// TIA Portal V19 export
FUNCTION "ValveMachine_PB_Connector" : Void   // FC157, LAD
TITLE = Collect push buttons for Valve Machine
// stored: Access Published, SetENOAutomatically false
   VAR_INPUT
      Enable : Bool;
      HMI_PB : "ValveMachine_PB";   // Push button from HMI a (e.g. MB1)
      LB_PB_Rest : Bool;
      LB_PB_Work : Bool;
      LB_PB_StartStop : Bool;
      Other_PB : "ValveMachine_PB";
   END_VAR
   VAR_OUTPUT
      PB : "ValveMachine_PB";
   END_VAR
BEGIN

REGION Network 1: Logical OR
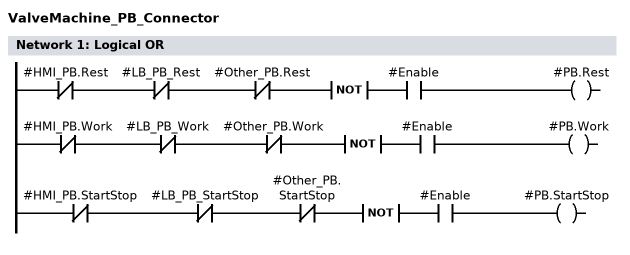
   RUNG wire#powerrail
      I_Contact( #HMI_PB.Rest )
      I_Contact( #LB_PB_Rest )
      I_Contact( #Other_PB.Rest )
      Not()
      Contact( #Enable )
      Coil( #PB.Rest )
   END_RUNG
   RUNG wire#powerrail
      I_Contact( #HMI_PB.Work )
      I_Contact( #LB_PB_Work )
      I_Contact( #Other_PB.Work )
      Not()
      Contact( #Enable )
      Coil( #PB.Work )
   END_RUNG
   RUNG wire#powerrail
      I_Contact( #HMI_PB.StartStop )
      I_Contact( #LB_PB_StartStop )
      I_Contact( #Other_PB.StartStop )
      Not()
      Contact( #Enable )
      Coil( #PB.StartStop )
   END_RUNG
   // the same network as SCL:
   #PB.Rest := NOT (NOT #HMI_PB.Rest AND NOT #LB_PB_Rest AND NOT #Other_PB.Rest) AND #Enable;
   #PB.Work := NOT (NOT #HMI_PB.Work AND NOT #LB_PB_Work AND NOT #Other_PB.Work) AND #Enable;
   #PB.StartStop := NOT (NOT #HMI_PB.StartStop AND NOT #LB_PB_StartStop AND NOT #Other_PB.StartStop) AND #Enable;
END_REGION
END_FUNCTION
